(* IEC 61131-3 sources: plc_generation_empirical_study/our_method_delta_DVP48ES300R/tests/fixtures/ladder, 1 file *)

(* ---- MotorControl.interface.st ---- *)
FUNCTION_BLOCK MotorControl
VAR_INPUT
    StartButton : BOOL;
    StopButton : BOOL;
    Permit : BOOL;
END_VAR
VAR_OUTPUT
    MotorRun : BOOL;
    Ready : BOOL;
END_VAR
END_FUNCTION_BLOCK
